// TIA Portal V17 export
// export: Created 2022-07-28T18:02:45.8280556Z, ExportSetting None, DisplayName Totally Integrated Automation Portal, DisplayVersion V17, DisplayName TIA Portal Openness, DisplayVersion V17, DisplayName TIA Portal Teamcenter Gateway, DisplayVersion V17, DisplayName TIA Portal Version Control Interface, DisplayVersion V17, DisplayName TIA Portal Test Suite Advanced, DisplayVersion V17, DisplayName SINAMICS Startdrive Advanced, DisplayVersion V17, DisplayName SINAMICS DCC, DisplayVersion V17, DisplayName SINAMICS Startdrive G130, G150, S120, S150, SINAMICS MV, S210, DisplayVersion V17, DisplayName SINAMICS Startdrive G110M, G120, G120C, G120D, G120P, G115D, DisplayVersion V17, DisplayName STEP 7 Professional, DisplayVersion V17, DisplayName SIMATIC Energy Suite, DisplayVersion V17, DisplayName STEP 7 CFC, DisplayVersion V17, DisplayName STEP 7 Safety, DisplayVersion V17, DisplayName WinCC Advanced / Unified PC, DisplayVersion V17, DisplayName SIMATIC Visualization Architect, DisplayVersion V17
FUNCTION_BLOCK "Lib_FB_Inverter_352Tel"   // FB287, SCL
TITLE = Communication via bus with inverter through telegram 352
{ S7_Optimized_Access := 'TRUE' }
AUTHOR : pngr
FAMILY : Bus
NAME : Tel352
// stored: AutoNumber false, MemoryReserve 100, SetENOAutomatically false
   VAR_INPUT
      I_ChangeDir : Bool := 0;   // Change direction
      II_Obj_ID : Int := -1;   // Technologie ID of current element
      I_HW_Tel_ID : HW_IO := 0;   // Hardware Identifer of telegram
   END_VAR
   VAR_OUTPUT
      Q_DataErr : Bool;   // 1 = Incorect data for read/write data to out DB
      Q_Error : Bool;
      QW_Status : Word := 0;   // Status output (7002 = FB in operation; 8xxx = error description - read the manual)
      QW_DiagId : Word := 16#0000;   // Error codes of the cyclic system funtion blocks DPWR / DPRD_DAT
   END_VAR
   VAR
      s_SendBuf : Struct   // Send buffer
         w_CTW1 : Word := WORD#16#0000;   // Control word
         w_SpeedSetpoint : Word := WORD#16#0000;   // Setpoint of speed
      END_STRUCT;
      s_RecvBuf : Struct   // Receive buffer
         w_STW1 : Word := WORD#16#0000;   // Status word
         w_SpeedActual : Word := WORD#16#0000;   // Actual speed
         w_ActualCurrent : Word;   // Actual current
         w_ActualTorque : Word;   // Actual torque
         w_Warning : Word;   // Warning code
         w_Fault : Word;   // Fault code
      END_STRUCT;
   END_VAR
   VAR_TEMP
      ti_RetSFC : Int;   // Status for fault analysis
      ti_Count : Int;   // Freely available counter variable 3
      tr_SpeedSP : Real;   // velocity
      tdw_RecvBuf : DWord;   // Buffer of Recv-Value
      tdw_SendBuf : DWord;   // Buffer of Send-Value
      t_LAddr : HW_IO;   // Start addr from the I/O process image area of mod (DEC) for DPWR_DAT/DPRD_DAT
      t_Obj_Any : DB_ANY;   // Ref to object data
      t_Obj_Var : Variant;   // Ref to object data
      t_DataErr : Bool;   // 1 = Transfer data error occured (ObjDB -> temp, ect)
      ti_NumObjDB : UInt;   // Number of DB for storage object data
      tui_DB_ShiftInv : UInt;
      t_InternalData : "Lib_UDT_Int";
      t_Obj_Inv : "Lib_UDT_Inverter_352Tel";
      t_SendBuf : Array[0..15] of Byte;   // Send buffer
      t_RecvBuf : Array[0..15] of Byte;   // Receive buffer
   END_VAR
BEGIN
   REGION Read data from output DB & reinit esential data
       //Set internal data
       "Lib_FC_GenMoto_InitInternal"(#t_InternalData);

       //Read Object data
       //Reinit temp values
       #t_Obj_Inv := "D_ZeroTypes".Inverter_352Tel;
       #tui_DB_ShiftInv := "D_General_ProgramDATA".ui_Shift_DB_Bus;

       IF #II_Obj_ID >= 0
       THEN
           //Read inverter data from output DB
           #ti_NumObjDB := INT_TO_UINT(#II_Obj_ID) + #tui_DB_ShiftInv;
           #t_Obj_Any := UINT_TO_DB_ANY(#ti_NumObjDB);
           #t_Obj_Var := DB_ANY_TO_VARIANT(in := #t_Obj_Any, err => #t_InternalData.i_Tmp);

           //If DB exist and convertion without error
           IF #t_InternalData.i_Tmp = 0
           THEN
               VariantGet(SRC := #t_Obj_Var,
                          DST => #t_Obj_Inv);
           ELSE
               #t_DataErr := true;
           END_IF;

       ELSE
           #t_DataErr := true;
       END_IF;

       //Reinit out values
       #Q_DataErr := false;
       #Q_Error := false;
       #QW_Status := w#16#0;
       #QW_DiagId := w#16#0;
   END_REGION
   //-------------------------------------------------------
   //-------------------------------------------------------
   IF NOT #t_DataErr
   THEN
       REGION Read data from Inverter and evaluate result
           // Try read data from inverter
           #ti_RetSFC := DPRD_DAT(LADDR := #I_HW_Tel_ID,
                                  RECORD => #t_RecvBuf);

           #QW_DiagId := INT_TO_WORD(#ti_RetSFC);

           //Evaluate result
           //If error occured
           IF #ti_RetSFC <> 0
           THEN
               //Reset bits in receive buffer
               FOR #ti_Count := 0 TO 11 DO
                   #t_RecvBuf[0] := b#16#0;
               END_FOR;

               //Set error
               #Q_Error := TRUE;
               #t_Obj_Inv.Read_WriteErr := TRUE;
               #QW_Status := 16#8600;

           ELSE// Read process was finish without error
               REGION Store bytes from buffer into word
                   #s_RecvBuf.w_STW1.%B0 := #t_RecvBuf[1];
                   #s_RecvBuf.w_STW1.%B1 := #t_RecvBuf[0];
                   #s_RecvBuf.w_SpeedActual.%B0 := #t_RecvBuf[3];
                   #s_RecvBuf.w_SpeedActual.%B1 := #t_RecvBuf[2];
                   #s_RecvBuf.w_ActualCurrent.%B0 := #t_RecvBuf[5];
                   #s_RecvBuf.w_ActualCurrent.%B1 := #t_RecvBuf[4];
                   #s_RecvBuf.w_ActualTorque.%B0 := #t_RecvBuf[7];
                   #s_RecvBuf.w_ActualTorque.%B1 := #t_RecvBuf[6];
                   #s_RecvBuf.w_Warning.%B0 := #t_RecvBuf[9];
                   #s_RecvBuf.w_Warning.%B1 := #t_RecvBuf[8];
                   #s_RecvBuf.w_Fault.%B0 := #t_RecvBuf[11];
                   #s_RecvBuf.w_Fault.%B1 := #t_RecvBuf[10];
               END_REGION
               //-------------------------------------------------------
               //-------------------------------------------------------
               REGION Store status word into bits
                   // Statement section REGION 
                   #t_Obj_Inv.Receive.STW.ReadyToSwitchOn := #s_RecvBuf.w_STW1.%X0;
                   #t_Obj_Inv.Receive.STW.ReadyToOperation := #s_RecvBuf.w_STW1.%X1;
                   #t_Obj_Inv.Receive.STW.OperationEnabled := #s_RecvBuf.w_STW1.%X2;
                   #t_Obj_Inv.Receive.STW.FaultActive := #s_RecvBuf.w_STW1.%X3;
                   #t_Obj_Inv.Receive.STW.OFF2Inactive := #s_RecvBuf.w_STW1.%X4;
                   #t_Obj_Inv.Receive.STW.OFF3Inactive := #s_RecvBuf.w_STW1.%X5;
                   #t_Obj_Inv.Receive.STW.LockoutActive := #s_RecvBuf.w_STW1.%X6;
                   #t_Obj_Inv.Receive.STW.AlarmActive := #s_RecvBuf.w_STW1.%X7;
                   #t_Obj_Inv.Receive.STW.SetpointReached := #s_RecvBuf.w_STW1.%X8;
                   #t_Obj_Inv.Receive.STW.CtrlRequest := #s_RecvBuf.w_STW1.%X9;
                   #t_Obj_Inv.Receive.STW.MaxSpeedReached := #s_RecvBuf.w_STW1.%X10;
                   #t_Obj_Inv.Receive.STW.IMP_LimitReached := #s_RecvBuf.w_STW1.%X11;
                   #t_Obj_Inv.Receive.STW.BrakeOpen := #s_RecvBuf.w_STW1.%X12;
                   #t_Obj_Inv.Receive.STW.Overtemperature := #s_RecvBuf.w_STW1.%X13;
                   #t_Obj_Inv.Receive.STW.ForwardBeckward := #s_RecvBuf.w_STW1.%X14;
                   #t_Obj_Inv.Receive.STW.PowerUnitOverload := #s_RecvBuf.w_STW1.%X15;
               END_REGION
               //-------------------------------------------------------
               //-------------------------------------------------------
               (* Vertion for new FW and TIA
                    SCATTER(IN := #s_RecvBuf.w_STW1,
                           OUT => #t_Obj_Inv.Receive.STW); *)

               //Set status if fault or lockout active
               IF #t_Obj_Inv.Receive.STW.FaultActive
               THEN
                   #QW_Status := 16#8401;
               ELSIF #t_Obj_Inv.Receive.STW.LockoutActive
               THEN
                   #QW_Status := 16#8402;
               ELSE
                   #QW_Status := 16#7002;
               END_IF;
               //-------------------------------------------------------
               //-------------------------------------------------------
               REGION Scalled actual values
                   //Speed
                   IF #t_Obj_Inv.Send.r_ReferenceSpeed <> 0.0
                   THEN
                       #t_Obj_Inv.Receive.r_ActualSpeed := INT_TO_REAL(WORD_TO_INT(#s_RecvBuf.w_SpeedActual)) / (16384.0 / #t_Obj_Inv.Send.r_ReferenceSpeed);
                   ELSE
                       #t_Obj_Inv.Receive.r_ActualSpeed := 0.0;
                   END_IF;

                   //If change dirrection
                   IF #I_ChangeDir
                   THEN
                       #t_Obj_Inv.Receive.r_ActualSpeed *= -1.0;
                   END_IF;

                   //Current 
                   IF #t_Obj_Inv.Send.r_ReferenceCurrent <> 0.0
                   THEN
                       #t_Obj_Inv.Receive.r_ActualCurrent := INT_TO_REAL(WORD_TO_INT(#s_RecvBuf.w_ActualCurrent)) / (16384.0 / #t_Obj_Inv.Send.r_ReferenceCurrent);
                   ELSE
                       #t_Obj_Inv.Receive.r_ActualCurrent := 0.0;
                   END_IF;

                   //Torque
                   IF #t_Obj_Inv.Send.r_ReferenceCurrent <> 0.0
                   THEN
                       #t_Obj_Inv.Receive.r_ActualTorque := INT_TO_REAL(WORD_TO_INT(#s_RecvBuf.w_ActualTorque)) / (16384.0 / #t_Obj_Inv.Send.r_ReferenceTorque);
                   ELSE
                       #t_Obj_Inv.Receive.r_ActualTorque := 0.0;
                   END_IF;

                   //Warnings
                   #t_Obj_Inv.Receive.w_Warning := #s_RecvBuf.w_Warning;

                   //Faults
                   #t_Obj_Inv.Receive.w_Fault := #s_RecvBuf.w_Fault;
               END_REGION
               //-------------------------------------------------------
               //-------------------------------------------------------
               //Detect dirrection of rotation
               #t_Obj_Inv.Receive.RunningForward := #t_Obj_Inv.Receive.r_ActualSpeed > 0.0
               AND #t_Obj_Inv.Receive.STW.ReadyToOperation;
               #t_Obj_Inv.Receive.RunningReverse := #t_Obj_Inv.Receive.r_ActualSpeed < 0.0
               AND #t_Obj_Inv.Receive.STW.ReadyToOperation;
               #t_Obj_Inv.Receive.Running := #t_Obj_Inv.Receive.STW.ReadyToOperation;
           END_IF;
       END_REGION
       //-------------------------------------------------------
       //-------------------------------------------------------
       REGION Write data into inverter and evaluate result
           //If read was finish without err
           IF #ti_RetSFC = 0
           THEN
               //-------------------------------------------------------
               //-------------------------------------------------------
               REGION Store control bits into word
                   #s_SendBuf.w_CTW1.%X0 := #t_Obj_Inv.Send.CTW.OFF1;
                   #s_SendBuf.w_CTW1.%X1 := #t_Obj_Inv.Send.CTW.OFF2;
                   #s_SendBuf.w_CTW1.%X2 := #t_Obj_Inv.Send.CTW.OFF3;
                   #s_SendBuf.w_CTW1.%X3 := #t_Obj_Inv.Send.CTW.EnableOperation;
                   #s_SendBuf.w_CTW1.%X4 := #t_Obj_Inv.Send.CTW.EnableRFG;
                   #s_SendBuf.w_CTW1.%X5 := #t_Obj_Inv.Send.CTW.FrozeRFG;
                   #s_SendBuf.w_CTW1.%X6 := #t_Obj_Inv.Send.CTW.EnableSetpoint;
                   #s_SendBuf.w_CTW1.%X7 := #t_Obj_Inv.Send.CTW.Acknowlege;
                   #s_SendBuf.w_CTW1.%X8 := #t_Obj_Inv.Send.CTW.Bit8_NotUsed;
                   #s_SendBuf.w_CTW1.%X9 := #t_Obj_Inv.Send.CTW.Bit9_NotUsed;
                   #s_SendBuf.w_CTW1.%X10 := #t_Obj_Inv.Send.CTW.CtrlByPLC;
                   #s_SendBuf.w_CTW1.%X11 := #t_Obj_Inv.Send.CTW.ChangeDir;
                   #s_SendBuf.w_CTW1.%X12 := #t_Obj_Inv.Send.CTW.Bit12_NotUsed;
                   #s_SendBuf.w_CTW1.%X13 := #t_Obj_Inv.Send.CTW.MOP_Up;
                   #s_SendBuf.w_CTW1.%X14 := #t_Obj_Inv.Send.CTW.MOP_Dwn;
                   #s_SendBuf.w_CTW1.%X15 := #t_Obj_Inv.Send.CTW.Bit15_NotUsed;
               END_REGION

               (*Vertion for new FW and TIA 
              GATHER(IN := #t_Obj_Inv.Send.CTW,
                      OUT => #s_SendBuf.w_CTW1); 
               *)
               //-------------------------------------------------------
               //-------------------------------------------------------
               // Scalled setpoint speed
               IF #t_Obj_Inv.Send.r_ReferenceSpeed <> 0
               THEN

                   #tr_SpeedSP := #t_Obj_Inv.Send.r_SetpointSpeed * (16384.0 / #t_Obj_Inv.Send.r_ReferenceSpeed);

                   //If change dirrection
                   IF #I_ChangeDir
                   THEN
                       #tr_SpeedSP *= -1.0;
                   END_IF;

                   // Limits
                   IF #tr_SpeedSP > 32767
                   THEN
                       #tr_SpeedSP := 32767;
                   ELSIF #tr_SpeedSP < -32768
                   THEN
                       #tr_SpeedSP := -32768;
                   END_IF;

                   #s_SendBuf.w_SpeedSetpoint := INT_TO_WORD(REAL_TO_INT(#tr_SpeedSP));

               ELSE
                   #s_SendBuf.w_SpeedSetpoint := W#16#0;
               END_IF;

               //Store words into send buffer
               #t_SendBuf[0] := #s_SendBuf.w_CTW1.%B1;
               #t_SendBuf[1] := #s_SendBuf.w_CTW1.%B0;
               #t_SendBuf[2] := #s_SendBuf.w_SpeedSetpoint.%B1;
               #t_SendBuf[3] := #s_SendBuf.w_SpeedSetpoint.%B0;

               //Reset bits in spare bytes
               FOR #ti_Count := 4 TO 11 DO
                   #t_SendBuf[#ti_Count] := b#16#0;
               END_FOR;

               //Call FC for write
               #ti_RetSFC := DPWR_DAT(LADDR := #I_HW_Tel_ID,
                                      RECORD := #t_SendBuf);

               //Process return value
               #QW_DiagId := INT_TO_WORD(#ti_RetSFC);

               //If was called with error
           ELSE
               //Set error
               #Q_Error := TRUE;
               #t_Obj_Inv.Read_WriteErr := TRUE;
               #QW_Status := 16#8601;
           END_IF;

       END_REGION
       //-------------------------------------------------------
       //-------------------------------------------------------
       REGION Write data into out DB
           VariantPut(SRC := #t_Obj_Inv,
                      DST := #t_Obj_Var);
       END_REGION
       //-------------------------------------------------------
       //-------------------------------------------------------
   END_IF;
   //-------------------------------------------------------
   //-------------------------------------------------------       
   #Q_DataErr := #t_DataErr;
   //Test text 17.02.2022
END_FUNCTION_BLOCK
